INTERFACE IAxis

METHOD M_Diag : BOOL
VAR_INPUT
END_VAR
VAR_OUTPUT
	bNcError 	: BOOL;
	bDrvError 	: BOOL;
	iNcErrorId	: UDINT;
END_VAR
END_METHOD

METHOD M_Enable : BOOL
VAR_INPUT
	bEnable 	: BOOL;
	fOverride	: LREAL;
END_VAR
END_METHOD

METHOD M_HardwareDiag : BOOL
VAR_INPUT
	bExecute : BOOL;
END_VAR
END_METHOD

METHOD M_HardwareReset : BOOL
VAR_INPUT
	bExecute : BOOL;
END_VAR
END_METHOD

{attribute 'InstanceVar'}
METHOD M_Move : BOOL
VAR_INPUT
	bExecute	: BOOL;
	eMoveCmd	: E_MoveCmd;
	fVelocity	: LREAL;
	fPosition	: LREAL;
END_VAR
END_METHOD

METHOD M_Reset : BOOL
VAR_INPUT
	bExecute 	: BOOL;
END_VAR
END_METHOD

END_INTERFACE

(* stored: Version 1.1.0.1, ProductVersion 3.1.4024.11
   Itf IAxis: Id {35584f32-17aa-4e46-a1af-ffe027546062}
   Method M_Diag: Id {90a113e1-86ef-4adb-bd82-c2199afc07da}
   Method M_Enable: Id {75ac69d7-0b36-49eb-8fbe-a94ee5d7f944}
   Method M_HardwareDiag: Id {50758a2e-8ae5-4613-b0e6-b714bfe03425}
   Method M_HardwareReset: Id {95904806-896b-4e75-b927-9e50f6095efc}
   Method M_Move: Id {5520acfb-9af7-4bba-8d3e-77cab2d9b2bb}
   Method M_Reset: Id {6322a45c-6b75-446a-9479-46b31ecb7546} *)
